// SIMATIC STEP 7 (V5.x) project sort box - turn table
// CPU: CPU 312
// station: Hardware
// station: SIMATIC 300(1)
// station: P_ADR_BUS
// program: S7 Program(1)

SYMBOL_TABLE
"at entry"	I 0.0	BOOL
"S1"	I 0.1	BOOL
"S2"	I 0.2	BOOL
"at TT entry"	I 0.3	BOOL
"at unload pos"	I 0.5	BOOL
"at front"	I 0.6	BOOL
"at right"	I 0.7	BOOL
"at left entry"	I 1.0	BOOL
"at right entry"	I 1.1	BOOL
"start"	I 1.3	BOOL
"stop"	I 1.4	BOOL
"at back"	I 1.6	BOOL
"loop marker"	M 0.0	BOOL
"empty"	M 0.1	BOOL
"conv 1"	Q 0.0	BOOL
"conv 2"	Q 0.1	BOOL
"TT conv left"	Q 0.2	BOOL
"TT conv right"	Q 0.3	BOOL
"turn table"	Q 0.4	BOOL
"left conv"	Q 0.5	BOOL
"right conv"	Q 0.6	BOOL
END_SYMBOL_TABLE

ORGANIZATION_BLOCK OB 1
TITLE = "Main Program Sweep (Cycle)"
VERSION : 0.1
VAR_TEMP
  OB1_EV_CLASS : BYTE ;	//Bits 0-3 = 1 (Coming event), Bits 4-7 = 1 (Event class 1)
  OB1_SCAN_1 : BYTE ;	//1 (Cold restart scan 1 of OB 1), 3 (Scan 2-n of OB 1)
  OB1_PRIORITY : BYTE ;	//Priority of OB Execution
  OB1_OB_NUMBR : BYTE ;	//1 (Organization block 1, OB1)
  OB1_RESERVED_1 : BYTE ;	//Reserved for system
  OB1_RESERVED_2 : BYTE ;	//Reserved for system
  OB1_PREV_CYCLE : INT ;	//Cycle time of previous OB1 scan (milliseconds)
  OB1_MIN_CYCLE : INT ;	//Minimum cycle time of OB1 (milliseconds)
  OB1_MAX_CYCLE : INT ;	//Maximum cycle time of OB1 (milliseconds)
  OB1_DATE_TIME : DATE_AND_TIME ;	//Date and time OB1 started
END_VAR
BEGIN
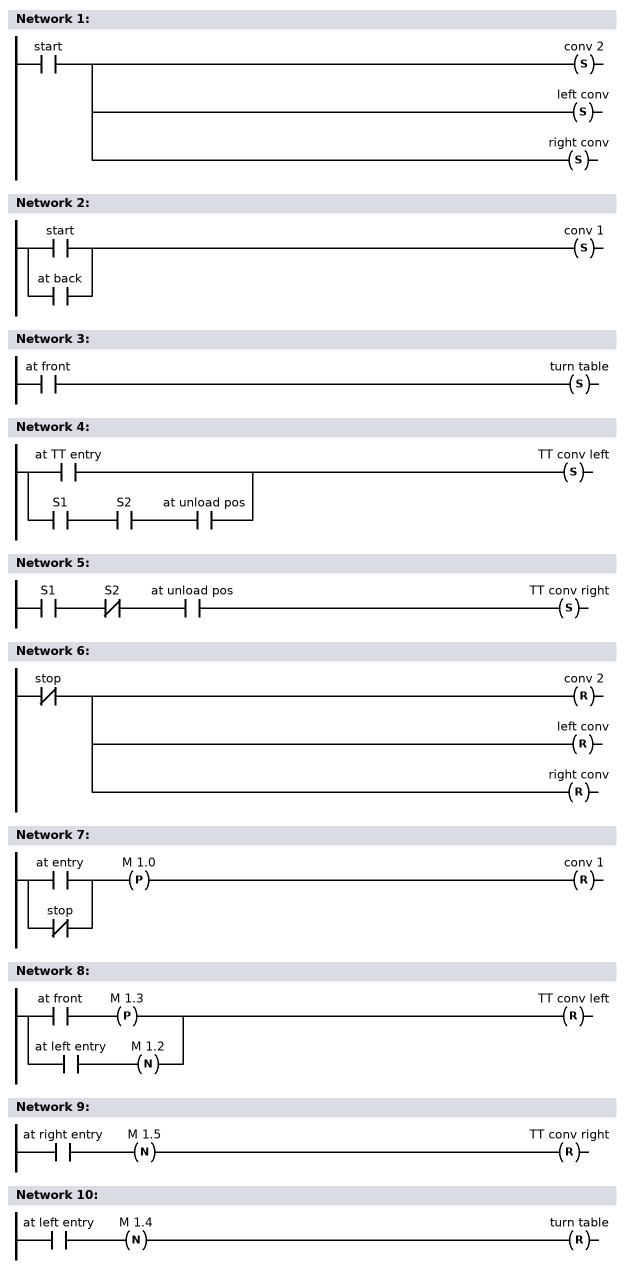
NETWORK
TITLE =
      A     "start";
      S     "conv 2";
      S     "left conv";
      S     "right conv";
NETWORK
TITLE =
      O     "start";
      O     "at back";
      S     "conv 1";
NETWORK
TITLE =
      A     "at front";
      S     "turn table";
NETWORK
TITLE =
      O     "at TT entry";
      O;
      A     "S1";
      A     "S2";
      A     "at unload pos";
      S     "TT conv left";
NETWORK
TITLE =
      A     "S1";
      AN    "S2";
      A     "at unload pos";
      S     "TT conv right";
NETWORK
TITLE =
      AN    "stop";
      R     "conv 2";
      R     "left conv";
      R     "right conv";
NETWORK
TITLE =
      A(;
      O     "at entry";
      ON    "stop";
      );
      FP    M 1.0;
      R     "conv 1";
NETWORK
TITLE =
      A     "at front";
      FP    M 1.3;
      O(;
      A     "at left entry";
      FN    M 1.2;
      );
      R     "TT conv left";
NETWORK
TITLE =
      A     "at right entry";
      FN    M 1.5;
      R     "TT conv right";
NETWORK
TITLE =
      A     "at left entry";
      FN    M 1.4;
      R     "turn table";
END_ORGANIZATION_BLOCK
